{attribute 'c++_compatible'}
FUNCTION_BLOCK FB_MyMqtt EXTENDS FB_IotMqttClient
VAR_INPUT
END_VAR
VAR_OUTPUT
END_VAR

VAR
	(* received message *)
	{attribute 'TcEncoding':='UTF-8'}
	sTopicRcv : STRING(255);
	{attribute 'TcEncoding':='UTF-8'}
	sPayloadRcv : STRING(255);
END_VAR

{attribute 'c++_compatible'}
{attribute 'pack_mode' := '4'}
{attribute 'show'}
{attribute 'minimal_input_size' := '4'}
METHOD OnMqttMessage : HRESULT
VAR_IN_OUT CONSTANT
	topic	: STRING;
END_VAR
VAR_INPUT
	payload	: PVOID;
	length	: UDINT;
	qos	: TcIotMqttQos;
	repeated	: BOOL;
END_VAR

VAR
	nPayloadRcvLen : UDINT;
END_VAR
SUPER^.nMessagesRcv := SUPER^.nMessagesRcv + 1;

STRNCPY( ADR(sTopicRcv), ADR(topic), SIZEOF(sTopicRcv) );             // important to use STRNCPY() to avoid an access to non-allocated memory
nPayloadRcvLen := MIN(length, DINT_TO_UDINT(SIZEOF(sPayloadRcv))-1);
MEMCPY( ADR(sPayloadRcv), payload, nPayloadRcvLen );
sPayloadRcv[nPayloadRcvLen] := 0;                                     // ensure a null termination of received string

OnMqttMessage := S_OK;
END_METHOD

END_FUNCTION_BLOCK

(* stored: Version 1.1.0.1, ProductVersion 3.1.4024.0
   POU FB_MyMqtt: Id {9c572ae6-e06d-4a20-9a98-0f29ff25b54f}, SpecialFunc None
   Method OnMqttMessage: Id {00b896c3-f44c-4cf4-aba5-b8400ecc5e1a} *)
